(* IEC 61131-3 sources: SRCI/RobotLibrarySysDep_Tc/Library/Memory, 3 files *)

(* ---- SysDepMemCmp.st ---- *)
/// System dependent implementation of the memory compare function
FUNCTION SysDepMemCmp : DINT
// -------------------------------------------------------------------------
//  SRCI Robot Library System Dependencies
// -------------------------------------------------------------------------
//
//  Object:      SysDepMemCmp
//  Author:      Thorsten Brach
//  Date:        2024-12-21
//
//  Description:
//    System specific implementation of the memory compare function.
//
//  Copyright:
//    (C) 2024 Thorsten Brach. All rights reserved
//             Licensed under the LGPL-3.0 license.
//
//  Disclaimer:
//    This project is provided without any guarantee and can be used for
//    private and commercial purposes. Any use is at the user’s
//    own risk and responsibility.
//
// -------------------------------------------------------------------------
VAR_INPUT
  /// Pointer to 1st memory area to be compared with the 2nd memory area
  pData1  : POINTER TO BYTE;
  /// Pointer to 2nd memory area to be compared with the 1st memory area
  pData2  : POINTER TO BYTE;
  /// Amount of bytes to be compared
  DataLen : UDINT;
END_VAR

  SysDepMemCmp := MemCmp( pBuf1 := pData1, pBuf2 := pData2, n := DataLen);

END_FUNCTION

(* ---- SysDepMemCpy.st ---- *)
/// System dependent implementation of the memory copy function
FUNCTION SysDepMemCpy : UDINT
// -------------------------------------------------------------------------
//  SRCI Robot Library System Dependencies
// -------------------------------------------------------------------------
//
//  Object:      SysDepMemCpy
//  Author:      Thorsten Brach
//  Date:        2024-12-21
//
//  Description:
//    System specific implementation of the memory copy function
//
//  Copyright:
//    (C) 2024 Thorsten Brach. All rights reserved
//             Licensed under the LGPL-3.0 license.
//
//  Disclaimer:
//    This project is provided without any guarantee and can be used for
//    private and commercial purposes. Any use is at the user’s
//    own risk and responsibility.
//
// -------------------------------------------------------------------------
VAR_INPUT
  /// Pointer to memory address to be copied to (target)
  pDest : POINTER TO BYTE;
  /// Pointer to memory address to be copied from (source)
  pSrc  : POINTER TO BYTE;
  /// Amount of bytes to be copied
  DataLen : UDINT;
END_VAR

  SysDepMemCpy := MemCpy( destAddr := pdest, srcAddr := pSrc, n := DataLen);

END_FUNCTION

(* ---- SysDepMemSet.st ---- *)
/// System dependent implementation of the memory set function
FUNCTION SysDepMemSet : UDINT
// -------------------------------------------------------------------------
//  SRCI Robot Library System Dependencies
// -------------------------------------------------------------------------
//
//  Object:      SysDepMemSet
//  Author:      Thorsten Brach
//  Date:        2024-12-21
//
//  Description:
//    System specific implementation of the memory set function
//
//  Copyright:
//    (C) 2024 Thorsten Brach. All rights reserved
//             Licensed under the LGPL-3.0 license.
//
//  Disclaimer:
//    This project is provided without any guarantee and can be used for
//    private and commercial purposes. Any use is at the user’s
//    own risk and responsibility.
//
// -------------------------------------------------------------------------
VAR_INPUT
  /// Pointer to memory address to be filled (target)
  pDest   : POINTER TO BYTE;
  /// Value with which the memory is to be initialized
  Value   : BYTE;
  /// Amount of bytes to be initialized in the memory block
  DataLen : UDINT;
END_VAR

  SysDepMemSet := MemSet( destAddr := pdest, fillByte := Value, n := DataLen);

END_FUNCTION
